TYPE ES_T5 :
	STRUCT
		Alarm			:ES_ALARM;
	
		S1_rt			:R_TRIG;	
		S1_letto		:BOOL;
	
	END_STRUCT
END_TYPE

(* stored: Version 1.1.0.1, ProductVersion 3.1.4022.6
   DUT ES_T5: Id {ab2be0df-f31f-4aaa-a54a-74b83ea907c1} *)
